PROGRAM sub_Heating
VAR
	fbVitramoBadOG		:	FB_Heating;
	
	fbFanGarage			:	FB_Fan;
	fbFanWerkstatt		:	FB_Fan;
END_VAR

//###################################################################################
//##-----------------------------------HEATING-------------------------------------##
//###################################################################################

//--------------------------------ENTFEUCHTER WERKSTATT------------------------
gvl_ea.bWOD01_3 := gvl_mb.Output_Coils[42];
//-----------------------------------------------------------------------------
//--------------------------------VITRAMO BAD----------------------------------
fbVitramoBadOG
(
	bInput			:=	gvl_EA.bID04_4,
	bInputOverwrite	:=	gvl_mb.Output_Coils[15],
	bOut			=>	gvl_EA.bOD04_4
);
//-----------------------------------------------------------------------------
//--------------------------------FAN Garage----------------------------------
fbFanGarage
(
	bInputControl	:=	gvl_EA.bWID01_14,
	bInputHA		:=	gvl_mb.Output_Coils[33],
	bOut			=>	gvl_EA.bWOD01_9,
	bOut			=>	gvl_mb.Output_Coils[33],
);
//-----------------------------------------------------------------------------
//--------------------------------FAN Werkstatt----------------------------------
fbFanWerkstatt
(
	bInputControl			:=	gvl_EA.bWID01_2,
	bLongPressControlled 	:=	TRUE,
	tLongPress				:=  T#1S,
	bInputHA				:=	gvl_mb.Output_Coils[26],
	bOut					=>	gvl_EA.bWOD01_4,
	bOut					=>	gvl_mb.Output_Coils[26],
);
//-----------------------------------------------------------------------------

END_PROGRAM

(* stored: Version 1.1.0.1, ProductVersion 3.1.4024.13
   POU sub_Heating: Id {2e634880-e46e-4912-9fc3-3ca3480f5766}, SpecialFunc None *)
